PROGRAM C11_OuterControlOACData
VAR

	fbMETSRestoreOCVData			: FB_OUTER_RestoreOCVDataFromStruct;
	fbWriteOACFileLoop				: FB_OUTER_WriteOACLoopDB;
	fbWriteErrorTable				: FB_OUTER_WriteErrorTable;
	fbFindErrorOuter				: FB_OUTER_FindErrorOuter;
	tofBarcodeFound				: TOF;

	sOACLastRecordDBName			: T_MaxString;

	(*rtMETSValidateOutersData		: R_TRIG;*)
	rtMETSRestoreOCVData		: R_TRIG;
	rtWriteOACFile				: R_TRIG;
	rtOACCounter				: R_TRIG;

	nErrorOuters					: UDINT;

	tonDisableRefeedButton			: TON;
	fbRepairOCVContent				: FB_OUTER_RepairOCVContentDB;

	fbFileWriteOACError				:FB_LOG_FileWriteError;
END_VAR

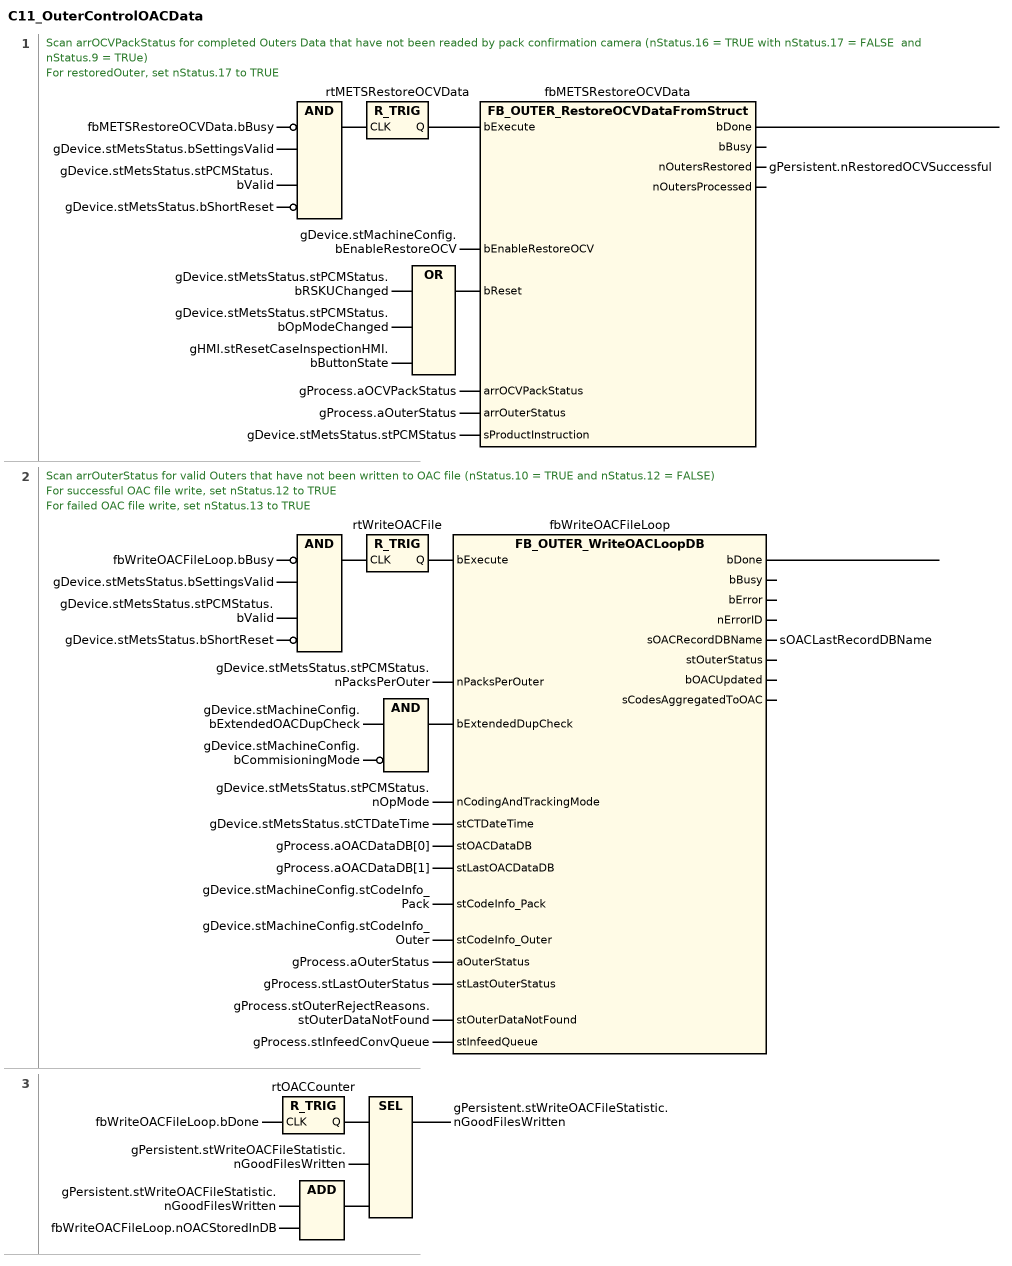
// NETWORK 1
// 					Scan arrOCVPackStatus for completed Outers Data that have not been readed by pack confirmation camera (nStatus.16 = TRUE with nStatus.17 = FALSE  and nStatus.9 = TRUe)
// For restoredOuter, set nStatus.17 to TRUE
//
//
rtMETSRestoreOCVData(CLK := NOT fbMETSRestoreOCVData.bBusy AND gDevice.stMetsStatus.bSettingsValid AND gDevice.stMetsStatus.stPCMStatus.bValid AND NOT gDevice.stMetsStatus.bShortReset); // R_TRIG
fbMETSRestoreOCVData(
    bExecute := rtMETSRestoreOCVData.Q,
    bEnableRestoreOCV := gDevice.stMachineConfig.bEnableRestoreOCV,
    bReset := gDevice.stMetsStatus.stPCMStatus.bRSKUChanged OR gDevice.stMetsStatus.stPCMStatus.bOpModeChanged OR gHMI.stResetCaseInspectionHMI.bButtonState,
    arrOCVPackStatus := gProcess.aOCVPackStatus,
    arrOuterStatus := gProcess.aOuterStatus,
    sProductInstruction := gDevice.stMetsStatus.stPCMStatus,
    nOutersRestored => gPersistent.nRestoredOCVSuccessful); // FB_OUTER_RestoreOCVDataFromStruct

// NETWORK 2
// 					Scan arrOuterStatus for valid Outers that have not been written to OAC file (nStatus.10 = TRUE and nStatus.12 = FALSE)
// For successful OAC file write, set nStatus.12 to TRUE
// For failed OAC file write, set nStatus.13 to TRUE
//
rtWriteOACFile(CLK := NOT fbWriteOACFileLoop.bBusy AND gDevice.stMetsStatus.bSettingsValid AND gDevice.stMetsStatus.stPCMStatus.bValid AND NOT gDevice.stMetsStatus.bShortReset); // R_TRIG
fbWriteOACFileLoop(
    bExecute := rtWriteOACFile.Q,
    nPacksPerOuter := gDevice.stMetsStatus.stPCMStatus.nPacksPerOuter,
    bExtendedDupCheck := gDevice.stMachineConfig.bExtendedOACDupCheck AND NOT gDevice.stMachineConfig.bCommisioningMode,
    nCodingAndTrackingMode := gDevice.stMetsStatus.stPCMStatus.nOpMode,
    stCTDateTime := gDevice.stMetsStatus.stCTDateTime,
    stOACDataDB := gProcess.aOACDataDB[0],
    stLastOACDataDB := gProcess.aOACDataDB[1],
    stCodeInfo_Pack := gDevice.stMachineConfig.stCodeInfo_Pack,
    stCodeInfo_Outer := gDevice.stMachineConfig.stCodeInfo_Outer,
    aOuterStatus := gProcess.aOuterStatus,
    stLastOuterStatus := gProcess.stLastOuterStatus,
    stOuterDataNotFound := gProcess.stOuterRejectReasons.stOuterDataNotFound,
    stInfeedQueue := gProcess.stInfeedConvQueue,
    sOACRecordDBName => sOACLastRecordDBName); // FB_OUTER_WriteOACLoopDB

// NETWORK 3
rtOACCounter(CLK := fbWriteOACFileLoop.bDone); // R_TRIG
gPersistent.stWriteOACFileStatistic.nGoodFilesWritten := SEL(rtOACCounter.Q, gPersistent.stWriteOACFileStatistic.nGoodFilesWritten, gPersistent.stWriteOACFileStatistic.nGoodFilesWritten + fbWriteOACFileLoop.nOACStoredInDB);

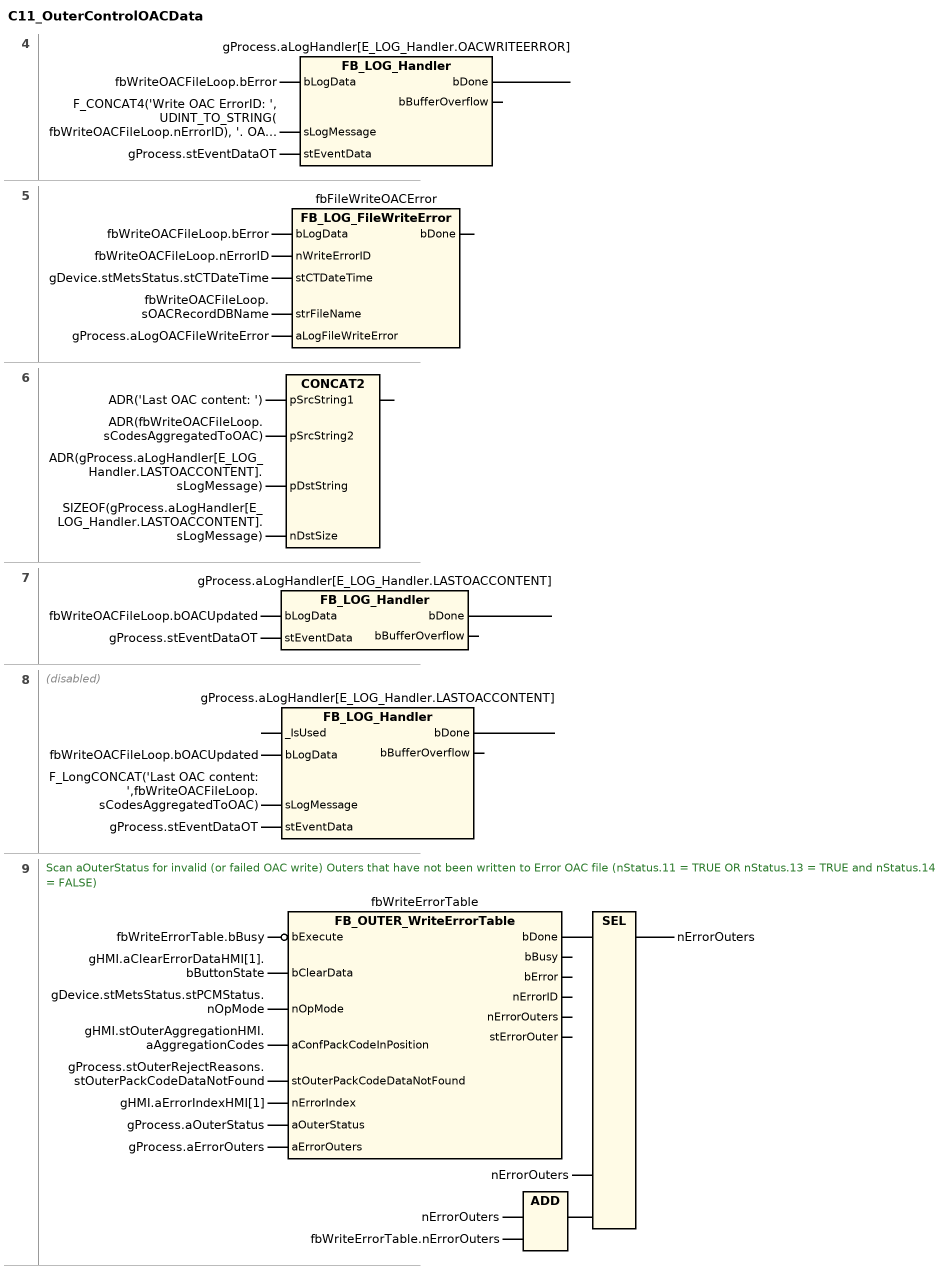
// NETWORK 4
gProcess.aLogHandler[E_LOG_Handler.OACWRITEERROR](
    bLogData := fbWriteOACFileLoop.bError,
    sLogMessage := F_CONCAT4('Write OAC ErrorID: ', UDINT_TO_STRING(fbWriteOACFileLoop.nErrorID), '. OAC File: ', fbWriteOACFileLoop.sOACRecordDBName),
    stEventData := gProcess.stEventDataOT); // FB_LOG_Handler

// NETWORK 5
fbFileWriteOACError(
    bLogData := fbWriteOACFileLoop.bError,
    nWriteErrorID := fbWriteOACFileLoop.nErrorID,
    stCTDateTime := gDevice.stMetsStatus.stCTDateTime,
    strFileName := fbWriteOACFileLoop.sOACRecordDBName,
    aLogFileWriteError := gProcess.aLogOACFileWriteError); // FB_LOG_FileWriteError

// NETWORK 6
CONCAT2(pSrcString1 := ADR('Last OAC content: '), pSrcString2 := ADR(fbWriteOACFileLoop.sCodesAggregatedToOAC), pDstString := ADR(gProcess.aLogHandler[E_LOG_Handler.LASTOACCONTENT].sLogMessage), nDstSize := SIZEOF(gProcess.aLogHandler[E_LOG_Handler.LASTOACCONTENT].sLogMessage));

// NETWORK 7
gProcess.aLogHandler[E_LOG_Handler.LASTOACCONTENT](bLogData := fbWriteOACFileLoop.bOACUpdated, stEventData := gProcess.stEventDataOT); // FB_LOG_Handler

// NETWORK 8 (disabled)
// gProcess.aLogHandler[E_LOG_Handler.LASTOACCONTENT](
//     bLogData := fbWriteOACFileLoop.bOACUpdated,
//     sLogMessage := F_LongCONCAT('Last OAC content: ',fbWriteOACFileLoop.sCodesAggregatedToOAC),
//     stEventData := gProcess.stEventDataOT); // FB_LOG_Handler

// NETWORK 9
// 					Scan aOuterStatus for invalid (or failed OAC write) Outers that have not been written to Error OAC file (nStatus.11 = TRUE OR nStatus.13 = TRUE and nStatus.14 = FALSE)
//
//
fbWriteErrorTable(
    bExecute := NOT fbWriteErrorTable.bBusy,
    bClearData := gHMI.aClearErrorDataHMI[1].bButtonState,
    nOpMode := gDevice.stMetsStatus.stPCMStatus.nOpMode,
    aConfPackCodeInPosition := gHMI.stOuterAggregationHMI.aAggregationCodes,
    stOuterPackCodeDataNotFound := gProcess.stOuterRejectReasons.stOuterPackCodeDataNotFound,
    nErrorIndex := gHMI.aErrorIndexHMI[1],
    aOuterStatus := gProcess.aOuterStatus,
    aErrorOuters := gProcess.aErrorOuters); // FB_OUTER_WriteErrorTable
nErrorOuters := SEL(fbWriteErrorTable.bDone, nErrorOuters, nErrorOuters + fbWriteErrorTable.nErrorOuters);

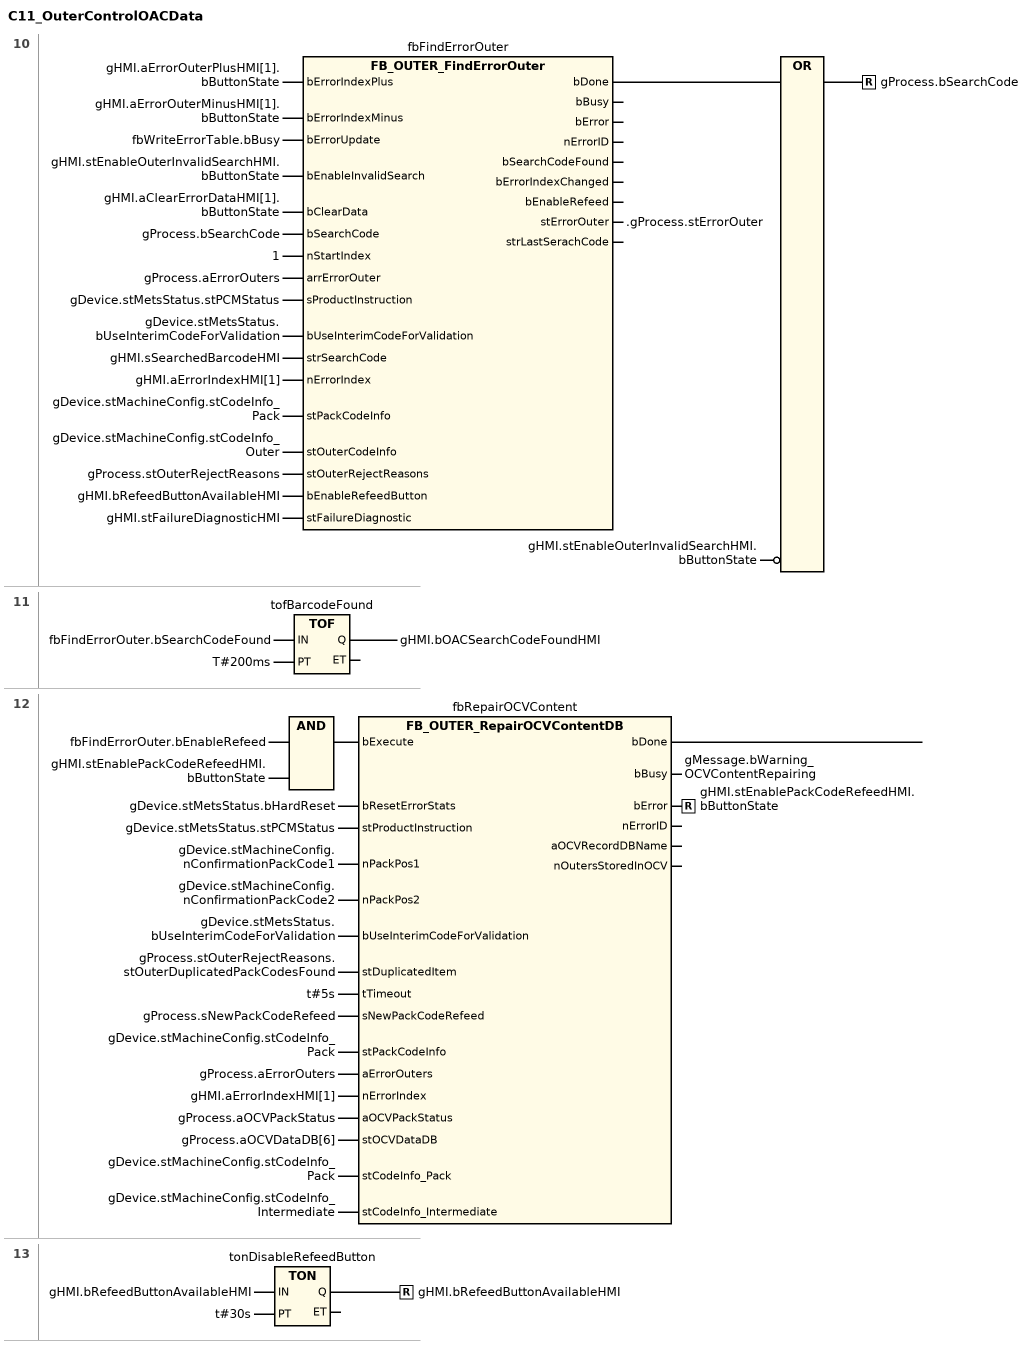
// NETWORK 10
fbFindErrorOuter(
    bErrorIndexPlus := gHMI.aErrorOuterPlusHMI[1].bButtonState,
    bErrorIndexMinus := gHMI.aErrorOuterMinusHMI[1].bButtonState,
    bErrorUpdate := fbWriteErrorTable.bBusy,
    bEnableInvalidSearch := gHMI.stEnableOuterInvalidSearchHMI.bButtonState,
    bClearData := gHMI.aClearErrorDataHMI[1].bButtonState,
    bSearchCode := gProcess.bSearchCode,
    nStartIndex := 1,
    arrErrorOuter := gProcess.aErrorOuters,
    sProductInstruction := gDevice.stMetsStatus.stPCMStatus,
    bUseInterimCodeForValidation := gDevice.stMetsStatus.bUseInterimCodeForValidation,
    strSearchCode := gHMI.sSearchedBarcodeHMI,
    nErrorIndex := gHMI.aErrorIndexHMI[1],
    stPackCodeInfo := gDevice.stMachineConfig.stCodeInfo_Pack,
    stOuterCodeInfo := gDevice.stMachineConfig.stCodeInfo_Outer,
    stOuterRejectReasons := gProcess.stOuterRejectReasons,
    bEnableRefeedButton := gHMI.bRefeedButtonAvailableHMI,
    stFailureDiagnostic := gHMI.stFailureDiagnosticHMI,
    stErrorOuter => .gProcess.stErrorOuter); // FB_OUTER_FindErrorOuter
gProcess.bSearchCode R= fbFindErrorOuter.bDone OR NOT gHMI.stEnableOuterInvalidSearchHMI.bButtonState;

// NETWORK 11
tofBarcodeFound(IN := fbFindErrorOuter.bSearchCodeFound, PT := T#200ms); // TOF
gHMI.bOACSearchCodeFoundHMI := tofBarcodeFound.Q;

// NETWORK 12
fbRepairOCVContent(
    bExecute := fbFindErrorOuter.bEnableRefeed AND gHMI.stEnablePackCodeRefeedHMI.bButtonState,
    bResetErrorStats := gDevice.stMetsStatus.bHardReset,
    stProductInstruction := gDevice.stMetsStatus.stPCMStatus,
    nPackPos1 := gDevice.stMachineConfig.nConfirmationPackCode1,
    nPackPos2 := gDevice.stMachineConfig.nConfirmationPackCode2,
    bUseInterimCodeForValidation := gDevice.stMetsStatus.bUseInterimCodeForValidation,
    stDuplicatedItem := gProcess.stOuterRejectReasons.stOuterDuplicatedPackCodesFound,
    tTimeout := t#5s,
    sNewPackCodeRefeed := gProcess.sNewPackCodeRefeed,
    stPackCodeInfo := gDevice.stMachineConfig.stCodeInfo_Pack,
    aErrorOuters := gProcess.aErrorOuters,
    nErrorIndex := gHMI.aErrorIndexHMI[1],
    aOCVPackStatus := gProcess.aOCVPackStatus,
    stOCVDataDB := gProcess.aOCVDataDB[6],
    stCodeInfo_Pack := gDevice.stMachineConfig.stCodeInfo_Pack,
    stCodeInfo_Intermediate := gDevice.stMachineConfig.stCodeInfo_Intermediate,
    bBusy => gMessage.bWarning_OCVContentRepairing); // FB_OUTER_RepairOCVContentDB
gHMI.stEnablePackCodeRefeedHMI.bButtonState R= fbRepairOCVContent.bError;

// NETWORK 13
tonDisableRefeedButton(IN := gHMI.bRefeedButtonAvailableHMI, PT := t#30s); // TON
gHMI.bRefeedButtonAvailableHMI R= tonDisableRefeedButton.Q;

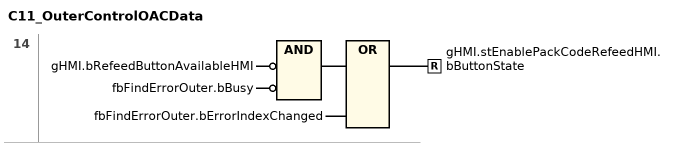
// NETWORK 14
gHMI.stEnablePackCodeRefeedHMI.bButtonState R= NOT gHMI.bRefeedButtonAvailableHMI AND NOT fbFindErrorOuter.bBusy OR fbFindErrorOuter.bErrorIndexChanged;

END_PROGRAM

(* stored: Version 1.1.0.1
   POU C11_OuterControlOACData: Id {bccc5893-30ae-41f5-bc97-08e06e6142bf}, SpecialFunc None *)
